Fanuc KAREL source: kt00371.KL

-- PROVISIONAL review KL for V1013-1; original PC SHA256 6c2074e0417f24690e675d6a1ed1af279765c712564de6c16f3f45c06b058bab
-- Incomplete behavior may be omitted. Consult companion uncertainty JSON. Do not deploy.
PROGRAM KT00371
%NOLOCKGROUP
VAR
  R1 : REAL
  OUT : BOOLEAN
-- UNRESOLVED_DECL Y2 type=002018
BEGIN
  -- UNRESOLVED_PC offsets 5-16; opcodes 2E,23
  -- UNRESOLVED_PC offsets 21-35; opcodes 2E,22,9D,33,B2
  -- UNRESOLVED_PC offsets 40-63; opcodes 21,22,9D,33,B1,64,70,23
  -- UNRESOLVED_PC offsets 68-72; opcodes 7F
END KT00371
